TYPE T_Ctrl_SIf_MDC_Ilk :
STRUCT
END_STRUCT
END_TYPE

(* stored: Version 1.1.0.1, ProductVersion 3.1.0.19
   DUT T_Ctrl_SIf_MDC_Ilk: Id {c54be6d4-af5e-4bf7-bcd9-68e6d5f94c74} *)
